// TIA Portal V18 export
// export: Created 2026-06-08T16:32:19.6793443Z, ExportSetting WithDefaults, DisplayName Totally Integrated Automation Portal, DisplayVersion V18, DisplayName TIA Portal Openness, DisplayVersion V18, DisplayName TIA Portal Version Control Interface, DisplayVersion V18, DisplayName STEP 7 Professional, DisplayVersion V18, DisplayName STEP 7 Safety, DisplayVersion V18, DisplayName WinCC Professional, DisplayVersion V18
VAR_GLOBAL   // PLC tag table "Assembly_tags"
   "Assembly green lid start" AT %I8.0 : Bool;
   "Assembly blue lid start" AT %I8.1 : Bool;
   "Assembly green base start" AT %I8.2 : Bool;
   "Assembly blue base start" AT %I8.3 : Bool;
   "G_lid in place" AT %I8.4 : Bool;
   "G_base in place" AT %I8.5 : Bool;
   G_lid_clamped AT %I8.6 : Bool;
   G_base_clamped AT %I8.7 : Bool;
   G_part_leaving AT %I9.0 : Bool;
   G_item_detect AT %I9.1 : Bool;
   "B_lid in place" AT %I9.2 : Bool;
   "B_base in place" AT %I9.3 : Bool;
   B_lid_clamped AT %I9.4 : Bool;
   B_base_clamped AT %I9.5 : Bool;
   B_part_leaving AT %I9.6 : Bool;
   B_item_detect AT %I9.7 : Bool;
   G_Negative_Trig_1 AT %M4.0 : Bool;
   G_Negative_Trig_2 AT %M4.1 : Bool;
   G_Negative_Trig_3 AT %M4.2 : Bool;
   move_green_lid_conv AT %M4.3 : Bool;
   move_green_base_conv AT %M4.4 : Bool;
   move_blue_lid_conv AT %M4.5 : Bool;
   move_blue_base_conv AT %M4.6 : Bool;
   B_Negative_Trig_1 AT %M4.7 : Bool;
   B_Negative_Trig_2 AT %M5.0 : Bool;
   B_Negative_Trig_3 AT %M5.1 : Bool;
   G_Detected_Memory AT %M5.2 : Bool;
   G_Reset AT %M5.3 : Bool;
   B_Detected_Memory AT %M5.4 : Bool;
   B_Reset AT %M5.5 : Bool;
   G_Timer_1 AT %T0 : Timer;
   G_Timer_2 AT %T1 : Timer;
   G_Timer_3 AT %T2 : Timer;
   B_Timer_1 AT %T3 : Timer;
   B_Timer_2 AT %T4 : Timer;
   B_Timer_3 AT %T5 : Timer;
   G_lids_conv_1 AT %Q7.0 : Bool;
   G_lids_conv_2 AT %Q7.1 : Bool;
   G_lids_conv_3 AT %Q7.2 : Bool;
   G_lids_conv_4 AT %Q7.3 : Bool;
   G_lids_conv_5 AT %Q7.4 : Bool;
   G_lids_conv_6 AT %Q7.5 : Bool;
   G_lids_conv_7 AT %Q7.6 : Bool;
   G_lids_conv_8 AT %Q7.7 : Bool;
   B_lids_conv_1 AT %Q8.0 : Bool;
   B_lids_conv_2 AT %Q8.1 : Bool;
   B_lids_conv_3 AT %Q8.2 : Bool;
   B_lids_conv_4 AT %Q8.3 : Bool;
   G_base_conv_1 AT %Q8.4 : Bool;
   G_base_conv_2 AT %Q8.5 : Bool;
   G_base_conv_3 AT %Q8.6 : Bool;
   G_base_conv_4 AT %Q8.7 : Bool;
   G_base_conv_5 AT %Q9.0 : Bool;
   G_base_conv_6 AT %Q9.1 : Bool;
   B_base_conv_1 AT %Q9.2 : Bool;
   B_base_conv_2 AT %Q9.3 : Bool;
   B_base_conv_3 AT %Q9.4 : Bool;
   B_base_conv_4 AT %Q9.5 : Bool;
   G_clamp_lid AT %Q9.6 : Bool;
   G_clamp_base AT %Q9.7 : Bool;
   "G_move Z" AT %Q10.0 : Bool;
   G_grab AT %Q10.1 : Bool;
   "G_move X" AT %Q10.2 : Bool;
   "G_pos.Raise_bases" AT %Q10.3 : Bool;
   B_clamp_lid AT %Q10.4 : Bool;
   B_clamp_base AT %Q10.5 : Bool;
   "B_move Z" AT %Q10.6 : Bool;
   B_grab AT %Q10.7 : Bool;
   "B_move X" AT %Q11.0 : Bool;
   "B_pos.Raise_bases" AT %Q11.1 : Bool;
END_VAR
